TYPE U_NCI_AXIS_ID_GROUP :
UNION

  stCtrl              : ARRAY[1..MAX_NCI_CH] OF ST_3D_Group;

  byCtrl    AT %q*    : ARRAY[1..MAX_NCI_CH] OF
                        ARRAY[1..SIZEOF(ST_3D_Group)] OF BYTE;
END_UNION
END_TYPE

(* stored: Version 1.1.0.1
   DUT U_NCI_AXIS_ID_GROUP: Id {aa4a6c2f-485a-4b5e-8de4-efbc39c8d21b} *)
